FUNCTION_BLOCK Directory EXTENDS Component
VAR
	children 			: ARRAY [1..Param.NumberOfChildren] OF I_Component;
	childCount			: INT := 0;
END_VAR

METHOD AddChild
VAR_INPUT
	Child : I_Component;
END_VAR


VAR
	i: INT;
END_VAR

childCount := childCount + 1;
children[childCount] := Child;
END_METHOD

METHOD GetChildren : ARRAY [1..Param.NumberOfChildren] OF I_Component;
GetChildren := children;
END_METHOD

PROPERTY GetSize : INT
GET
VAR
	i : INT := 0;
END_VAR
FOR i := 1 TO childCount  DO	
	GetSize := GetSize + children[i].GetSize;
END_FOR
END_GET
END_PROPERTY

METHOD ResetSize
childCount:= 0;
END_METHOD

END_FUNCTION_BLOCK

(* stored: Version 1.1.0.1, ProductVersion 3.1.4024.12
   POU Directory: Id {00d5b3f4-cd2a-48d7-a009-09c4bd5e016b}, SpecialFunc None
   Method AddChild: Id {742d5baf-9a6f-47dd-90fa-9711c41b74af}
   Method GetChildren: Id {b3c695ad-4f4a-45f6-92b2-b17c793b03e6}
   Property GetSize: Id {277022a1-2ddc-485d-b014-e9d2bb317b28}
   Get Get: Id {8798b121-fcac-450f-975a-514d46ada92d}
   Method ResetSize: Id {95e8d98d-a920-4d8f-b1f5-89ba0cefb3ac} *)
